{attribute 'linkalways'} 
{attribute 'no_explicit_call' := 'This FB is a CLASS and must be accessed using methods or properties'}
{attribute 'enable_dynamic_creation'}
FUNCTION_BLOCK _TcVnVector3_REAL EXTENDS AliasDatatypeBase
VAR
	localData : TcVnVector3_REAL;
	activeData : REFERENCE TO TcVnVector3_REAL REF= localData;
	aliasBaseDatatype : _Array0to2OfREAL;
END_VAR

PROPERTY PUBLIC Address : PVOID
GET
Address := ADR(activeData);
END_GET
END_PROPERTY

METHOD PUBLIC ClearReference
VAR_INPUT
END_VAR
activeData REF= localData;
SetBaseDatatypeReference();
END_METHOD

METHOD PUBLIC Clone : I_Datatype
VAR
    pClone : POINTER TO _TcVnVector3_REAL;
END_VAR
pClone := __NEW(_TcVnVector3_REAL);
Clone := pClone^;
END_METHOD

METHOD FB_init : BOOL
VAR_INPUT
	bInitRetains : BOOL; // if TRUE, the retain variables are initialized (warm start / cold start)
	bInCopyCode : BOOL;  // if TRUE, the instance afterwards gets moved into the copy code (online change)
	//InitialValue : <type>; // if possible, not all values can be initialized
END_VAR
//localData := InitialValue; // if possible, not all values can be initialized
SetBaseDatatypeReference();
AddBaseDatatype(aliasBaseDatatype);
END_METHOD

PROPERTY PUBLIC Identifier : T_MAXSTRING
GET
Identifier := 'TcVnVector3_REAL';
END_GET
END_PROPERTY

METHOD PUBLIC MakeReferenceTo
VAR_INPUT
	ReferenceTarget : REFERENCE TO TcVnVector3_REAL;
END_VAR
activeData REF= ReferenceTarget;
SetBaseDatatypeReference();
END_METHOD

METHOD PROTECTED SetBaseDatatypeReference
VAR_INPUT
END_VAR
aliasBaseDatatype.MakeReferenceTo(activeData);
END_METHOD

PROPERTY PUBLIC Size : UDINT
GET
Size := SIZEOF(activeData);
END_GET
END_PROPERTY

METHOD TryMakeReferenceTo : BOOL
VAR_INPUT
	Target : I_Datatype;
END_VAR
VAR
	pTargetData : POINTER TO TcVnVector3_REAL;
END_VAR
IF NOT IsEquivalentTo(Target) THEN
	RETURN;
END_IF

pTargetData := Target.Address;
activeData REF= pTargetData^;
SetBaseDatatypeReference();
TryMakeReferenceTo := TRUE;
END_METHOD

PROPERTY PUBLIC Value : REFERENCE TO TcVnVector3_REAL
GET
Value REF= activeData;
END_GET
END_PROPERTY

END_FUNCTION_BLOCK

(* stored: Version 1.1.0.1, ProductVersion 3.1.4024.13
   POU _TcVnVector3_REAL: Id {b3dab101-e7ed-0b0d-3cd1-6dfcc29c4cfe}, SpecialFunc None
   Folder Core: Id {e2cdb446-3584-0e93-39fb-baa8e1c9c4c2}
   Folder Protected: Id {9d5bae6a-a000-0704-1ed2-8e3b208f9723}
   Folder Customize: Id {dae0f781-9b65-0043-22cd-b7e9fe99f65a}
   Folder Constructor: Id {a167f21b-8ba9-085b-0fe4-5204f525ae90}
   Property Address: Id {91ac5f59-5176-0ac8-3348-d9b91b248180}
   Get Get: Id {27fb894f-60f8-0a1b-0224-a4dc2c93de41}
   Method ClearReference: Id {527fe126-b0a4-02a4-1c5d-1ec85e5f391d}
   Method Clone: Id {5c8f2ffe-ab42-0b74-020c-adbfef0af24f}
   Method FB_init: Id {ae108e70-3df1-07c0-1812-f68360d4b12a}
   Property Identifier: Id {3248cfaa-48bf-0d74-1d72-4dd23587fa3d}
   Get Get: Id {c4e14feb-667e-0515-0949-174b1dc6c3e5}
   Method MakeReferenceTo: Id {c065cc03-6812-0583-231e-e09a181d398a}
   Method SetBaseDatatypeReference: Id {30e53843-b7e5-0b40-01e2-9214d984494d}
   Property Size: Id {5d696c90-a0b3-004d-19a5-ee0492b53244}
   Get Get: Id {0d75c7e4-5f5a-0674-3cf0-e580ce1db700}
   Method TryMakeReferenceTo: Id {48253c0a-4f82-0b9e-1ca5-6d6afad81ba2}
   Property Value: Id {11fd3dbd-9417-0077-06fa-8887c2f6ed76}
   Get Get: Id {81c02776-a47c-052d-0d1c-99ee3f1d3a84} *)
